(* PLC project Programme MGS_v0.4.15_PlcTestsFramework_TranslationSuite.project, CODESYS CODESYS V3.5 SP19 Patch 1 *)
(* stored: creationDateTime 2026-07-17T01:20:50.7765012, modificationDateTime 2026-07-17T01:19:18.6752618 *)

FUNCTION_BLOCK FB_TestReference
  VAR
    refTest : REFERENCE TO FB_Winch;  (* n'importe quel FB existant suffit *)
  END_VAR

            
          
END_FUNCTION_BLOCK
